{attribute addProperty BoxType "IL2302-B110-0017"}
{attribute addProperty Id "Term_24KL_5BCCED4C00Term_395_Ix1000KL_9BB4615400"}
{attribute addProperty CRC "2094233823"}
{attribute addProperty SizeInBites "0"}
{attribute addProperty SizeInBytes "0"}
TYPE A_0024_IL2302_B110_0017_7CD378DF EXTENDS IL2302_4487A81F :
STRUCT
	{attribute addProperty Name "Term_24"}
	Term_24 : KL_5BCCED4C;
	{attribute addProperty Name "Term_395_Ix1000"}
	Term_395_Ix1000 : KL_9BB46154;
END_STRUCT
END_TYPE

(* stored: Version 1.2.0.0, ProductVersion 3.1.4024.9
   DUT A_0024_IL2302_B110_0017_7CD378DF: Id {7f5ee0a6-7b20-4c10-86b5-d24f30dc8a68} *)
